(* IEC 61131-3 sources: YaoKangDeviceDemo/src/50_FB, 7 files *)

(* ---- FC_DefaultAxisConfig.st ---- *)
(*============================================================================
  FC_DefaultAxisConfig —— 单轴限位/运动配置工厂默认（P5）
  ----------------------------------------------------------------------------
  返回 Stru_AxisLimitConfig 出厂值。三轴共用同一保守默认，现场按轴调试。
  ⚠ diPulsePerDeg 脉冲当量为占位，必须按 M900 电子齿轮/机械传动比核定后 Save。
==========================================================================*)
FUNCTION FC_DefaultAxisConfig : Stru_AxisLimitConfig

FC_DefaultAxisConfig.rPosLimit     := 90.0;     (* 正限位 ° *)
FC_DefaultAxisConfig.rNegLimit     := -90.0;    (* 负限位 ° *)
FC_DefaultAxisConfig.rInitPos      := 0.0;      (* 初始位置 ° *)
FC_DefaultAxisConfig.rTolerance    := 0.5;      (* 到位容差 ° *)
FC_DefaultAxisConfig.rMaxVel       := 50.0;     (* 最大速度 °/s *)
FC_DefaultAxisConfig.rMinVel       := 0.5;      (* 最小速度 °/s *)
FC_DefaultAxisConfig.rMaxAcc       := 100.0;    (* 最大加速度 °/s² *)
FC_DefaultAxisConfig.rMaxDec       := 100.0;    (* 最大减速度 °/s² *)
FC_DefaultAxisConfig.diPulsePerDeg := 10000;    (* 脉冲当量 Pulse/°（占位，待核定） *)
FC_DefaultAxisConfig.diTimeout     := 30000;    (* 定位超时 ms *)

END_FUNCTION

(* ---- FC_DefaultConditionParams.st ---- *)
(*============================================================================
  FC_DefaultConditionParams —— 调理参数工厂默认（P5）
  ----------------------------------------------------------------------------
  返回一整套 Stru_CondParams 出厂值（三轴 16 段往复 + 全局）。
  ⚠ 默认值仅为安全可校验的保守占位，现场须由工程师按工艺调试后 Save。
  单位：位置 °（脉冲当量见轴 Config）、速度 °/s、加减速 °/s²、时间 ms。
==========================================================================*)
FUNCTION FC_DefaultConditionParams : Stru_CondParams

(*--- 扭腰 SeatTwist：默认单段 ±10°、2 °/s、1 循环 ---*)
FC_DefaultConditionParams.SeatTwist.rAcc             := 20.0;
FC_DefaultConditionParams.SeatTwist.rDec             := 20.0;
FC_DefaultConditionParams.SeatTwist.rInitialPosition := 0.0;
FC_DefaultConditionParams.SeatTwist.iVelocityMode    := 0;
FC_DefaultConditionParams.SeatTwist.iCycleModeLen    := 1;
FC_DefaultConditionParams.SeatTwist.iCycleCount      := -1;
FC_DefaultConditionParams.SeatTwist.iSignalMode      := -1;
FC_DefaultConditionParams.SeatTwist.iSegmentCount    := 1;
FC_DefaultConditionParams.SeatTwist.bEnabled         := TRUE;
FC_DefaultConditionParams.SeatTwist.bOneWay          := FALSE;
FC_DefaultConditionParams.SeatTwist.arPosition[1]    := 10.0;
FC_DefaultConditionParams.SeatTwist.arVelocity[1]    := 2.0;
FC_DefaultConditionParams.SeatTwist.abCycleMode[1]   := FALSE;

(*--- 摆腿 LegAngle：默认单段 +15° ---*)
FC_DefaultConditionParams.LegAngle.rAcc             := 20.0;
FC_DefaultConditionParams.LegAngle.rDec             := 20.0;
FC_DefaultConditionParams.LegAngle.rInitialPosition := 0.0;
FC_DefaultConditionParams.LegAngle.iVelocityMode    := 0;
FC_DefaultConditionParams.LegAngle.iCycleModeLen    := 1;
FC_DefaultConditionParams.LegAngle.iCycleCount      := -1;
FC_DefaultConditionParams.LegAngle.iSignalMode      := -1;
FC_DefaultConditionParams.LegAngle.iSegmentCount    := 1;
FC_DefaultConditionParams.LegAngle.bEnabled         := TRUE;
FC_DefaultConditionParams.LegAngle.bOneWay          := FALSE;
FC_DefaultConditionParams.LegAngle.arPosition[1]    := 15.0;
FC_DefaultConditionParams.LegAngle.arVelocity[1]    := 3.0;
FC_DefaultConditionParams.LegAngle.abCycleMode[1]   := FALSE;

(*--- 冲击 ChestImpact：默认单段 +5°、较快 5 °/s ---*)
FC_DefaultConditionParams.ChestImpact.rAcc             := 30.0;
FC_DefaultConditionParams.ChestImpact.rDec             := 30.0;
FC_DefaultConditionParams.ChestImpact.rInitialPosition := 0.0;
FC_DefaultConditionParams.ChestImpact.iVelocityMode    := 0;
FC_DefaultConditionParams.ChestImpact.iCycleModeLen    := 1;
FC_DefaultConditionParams.ChestImpact.iCycleCount      := -1;
FC_DefaultConditionParams.ChestImpact.iSignalMode      := -1;
FC_DefaultConditionParams.ChestImpact.iSegmentCount    := 1;
FC_DefaultConditionParams.ChestImpact.bEnabled         := TRUE;
FC_DefaultConditionParams.ChestImpact.bOneWay          := FALSE;
FC_DefaultConditionParams.ChestImpact.arPosition[1]    := 5.0;
FC_DefaultConditionParams.ChestImpact.arVelocity[1]    := 5.0;
FC_DefaultConditionParams.ChestImpact.abCycleMode[1]   := FALSE;

(*--- 全局 ---*)
FC_DefaultConditionParams.rPusherPos       := 0.0;      (* 成角目标 °（尾板） *)
FC_DefaultConditionParams.rPusherInitPos   := 0.0;
FC_DefaultConditionParams.diBatchCount     := 1;        (* 老化批次数 *)
FC_DefaultConditionParams.diBatchInterval  := 5000;     (* 批次间隔 ms *)
FC_DefaultConditionParams.diTotalTimeout   := 300000;   (* 总超时 5 min *)
FC_DefaultConditionParams.diConfirmTimeout := 30000;    (* 确认超时 30 s *)
FC_DefaultConditionParams.iCycleCount      := 1;        (* 全局循环次数 *)
FC_DefaultConditionParams.iSignalMode      := 0;        (* 0=脚踏 1=自动 *)

END_FUNCTION

(* ---- FC_DefaultHomingParams.st ---- *)
(*============================================================================
  FC_DefaultHomingParams —— 回零参数工厂默认（P5）
  ----------------------------------------------------------------------------
  返回 Stru_HomingParams 出厂值（普通回零 + 紧急回零 Jog/防夹时序）。
  单位：速度 °/s、加减速 °/s²、扭矩 %、时间 ms。
==========================================================================*)
FUNCTION FC_DefaultHomingParams : Stru_HomingParams

(*--- 限位脱离 ---*)
FC_DefaultHomingParams.rLimitEscapeVel := 2.0;
(*--- 三轴 Jog 速度（内部轴序 1=Chest 2=Seat 3=Leg） ---*)
FC_DefaultHomingParams.rChestJogVel    := 5.0;
FC_DefaultHomingParams.rSeatJogVel     := 5.0;
FC_DefaultHomingParams.rLegJogVel      := 5.0;
(*--- 三轴接近微调（爬行）速度 ---*)
FC_DefaultHomingParams.rChestCrawlVel  := 0.5;
FC_DefaultHomingParams.rSeatCrawlVel   := 0.5;
FC_DefaultHomingParams.rLegCrawlVel    := 0.5;
(*--- 接近区（进入后切爬行） ---*)
FC_DefaultHomingParams.rChestApproachZone := 3.0;
FC_DefaultHomingParams.rSeatApproachZone  := 3.0;
FC_DefaultHomingParams.rLegApproachZone   := 3.0;
(*--- 到位迟滞窗口 ---*)
FC_DefaultHomingParams.rChestHysteresis := 0.3;
FC_DefaultHomingParams.rSeatHysteresis  := 0.3;
FC_DefaultHomingParams.rLegHysteresis   := 0.3;
(*--- Jog 加速度 ---*)
FC_DefaultHomingParams.rChestJogAcc := 20.0;
FC_DefaultHomingParams.rSeatJogAcc  := 20.0;
FC_DefaultHomingParams.rLegJogAcc   := 20.0;
(*--- 防夹扭矩限（净扭矩 %，紧急回零 Jog 超阈即停重试） ---*)
FC_DefaultHomingParams.rAntiPinchTorqueLimit := 40.0;
(*--- 超时/时序 ---*)
FC_DefaultHomingParams.diHomingTimeout         := 60000;   (* 普通回零全流程 60 s *)
FC_DefaultHomingParams.diEmergencyTimeout      := 30000;   (* 紧急回零 30 s *)
FC_DefaultHomingParams.diLimitEscapeTimeout    := 10000;   (* 限位脱离 10 s *)
FC_DefaultHomingParams.diStopReleaseTimeout    := 5000;    (* MC_Stop 释放等待 5 s *)
FC_DefaultHomingParams.diEmergencyCoastMs      := 500;     (* 停后滑行等待 *)
FC_DefaultHomingParams.diEmergencyStallTimeout := 2000;    (* 防夹堵转判定 2 s *)
(*--- 模式/重试 ---*)
FC_DefaultHomingParams.iHomingMode          := 0;         (* 0=顺序 1=并行（默认顺序） *)
FC_DefaultHomingParams.iMaxRetry            := 3;         (* 防夹重试上限 *)
FC_DefaultHomingParams.bEmergencyAllowCalib := FALSE;     (* 紧急回零默认不触发标定 *)

END_FUNCTION

(* ---- FC_DefaultPusherConfig.st ---- *)
(*============================================================================
  FC_DefaultPusherConfig —— 电推杆（尾板）配置工厂默认（P5）
  ----------------------------------------------------------------------------
  返回 Stru_PusherLimitConfig 出厂值：开关型电推杆 + HC_Counter(mm) + 几何解算，
  全部角度阈值直接以 ° 为单位（无脉冲/AD 字段）；堵转/超时/换向缓冲/软限位保留。
  ⚠ 角度°阈值（rMinTravel/rInertiaUp/Down/rStallThreshold）为占位，
    必须现场调试后 Save；几何长度/补偿常量在 GVL_CONST（PUSHER_GEO_*）。
==========================================================================*)
FUNCTION FC_DefaultPusherConfig : Stru_PusherLimitConfig

FC_DefaultPusherConfig.rMaxDeg              := 80.0;     (* 正限位 ° *)
FC_DefaultPusherConfig.rMinDeg              := 0.0;      (* 负限位 ° *)
FC_DefaultPusherConfig.rTolerance           := 0.5;      (* 到位容差 ° *)
FC_DefaultPusherConfig.rInitialPosition     := 0.0;      (* 初始位置（回零目标）° *)
FC_DefaultPusherConfig.rMinTravel           := 2.0;      (* 堵转检测前最小行程 °（占位） *)
FC_DefaultPusherConfig.rHomePosition        := 0.0;      (* 原点位置 ° *)
FC_DefaultPusherConfig.rInertiaUp           := 1.0;      (* 角度增大向惯性补偿 °（占位） *)
FC_DefaultPusherConfig.rInertiaDown         := 1.0;      (* 角度减小向惯性补偿 °（占位） *)
FC_DefaultPusherConfig.rStallThreshold      := 0.5;      (* 堵转位移阈值 °（占位） *)
FC_DefaultPusherConfig.rStallSpeedThreshold := 0.5;      (* 堵转速度阈值 °/s（占位） *)
FC_DefaultPusherConfig.diStallTimeout       := 1000;     (* 堵转判定 1 s *)
FC_DefaultPusherConfig.diTimeout            := 30000;    (* 寻传感器/标定 30 s *)
FC_DefaultPusherConfig.diReverseDelay       := 500;      (* 换向缓冲 0.5 s *)
FC_DefaultPusherConfig.diStopCheck          := 500;      (* 停车滑行等待 0.5 s *)
FC_DefaultPusherConfig.iMaxRetries          := 3;        (* 最大修正次数 *)
FC_DefaultPusherConfig.bInvertPusherDirection := FALSE;  (* 输出方向不取反 *)

END_FUNCTION

(* ---- FC_ValidateParams.st ---- *)
(*============================================================================
  FC_ValidateParams —— 参数 Apply 前校验（P5）
  ----------------------------------------------------------------------------
  对指定参数块的编辑缓冲（HMI 区）做合法性检查，非法即拒绝且不触碰运行区。
  入参：iBlock —— 1=Condition 调理参数（含三轴 16 段往复）
                  2=Pusher 推杆配置（iErrAxis 恒为 AXIS_ID_TAIL=4）
                  3=Chest 冲击轴 Config（iErrAxis=1）
                  4=Leg   转角轴 Config（iErrAxis=2）
                  5=Seat  扭角轴 Config（iErrAxis=3）
                  6=Homing 回零参数（iErrAxis=0，全局）
  出参：iErrCode  —— 0=通过；PARAM_ERR_SEGMENT=1005 段数非法；ERR_PARAM_VALUE=5007 值非法
        iErrAxis  —— 错误所在轴（1=Chest 2=Leg 3=Seat 4=Tail，0=全局）
        iErrField —— 错误字段索引（块内编号，随 iParamErrorField 上报 HMI 定位）
  返回：TRUE=校验通过可 Apply；FALSE=拒绝（三元组已填）。
  说明：仅静态范围/逻辑校验；跨块一致性（如段位置 vs 轴软限位）在运行前检查
       （7xxx，P10）兜底。范围阈值为保守工程值，现场可按工艺收紧。
==========================================================================*)
FUNCTION FC_ValidateParams : BOOL
VAR_INPUT
    iBlock      : INT;
END_VAR
VAR_OUTPUT
    iErrCode    : INT;
    iErrAxis    : INT;
    iErrField   : INT;
END_VAR
(* 段循环下标 vpI 与轴配置视图 vpCfg 为函数私有工作变量，H5U 不支持 FUNCTION 局部
   VAR，已上移为 GVL_Internal 全局（vpI:INT / vpCfg:Stru_AxisLimitConfig）。 *)

(* 默认通过 *)
FC_ValidateParams := TRUE;
iErrCode  := 0;
iErrAxis  := 0;
iErrField := 0;

(*==========================================================================
  iBlock = 1：调理参数（三轴往复 + 全局）
  ==========================================================================*)
IF iBlock = 1 THEN
    (*--- 扭腰 SeatTwist（iErrAxis=AXIS_ID_SEAT=3） ---*)
    IF HMI.Condition.Param.SeatTwist.bEnabled THEN
        IF (HMI.Condition.Param.SeatTwist.iSegmentCount < 1) OR
           (HMI.Condition.Param.SeatTwist.iSegmentCount > 16) THEN
            FC_ValidateParams := FALSE; iErrCode := PARAM_ERR_SEGMENT; iErrAxis := AXIS_ID_SEAT; iErrField := 1; RETURN;
        END_IF;
        IF HMI.Condition.Param.SeatTwist.rAcc <= 0.0 THEN
            FC_ValidateParams := FALSE; iErrCode := ERR_PARAM_VALUE; iErrAxis := AXIS_ID_SEAT; iErrField := 2; RETURN;
        END_IF;
        IF HMI.Condition.Param.SeatTwist.rDec <= 0.0 THEN
            FC_ValidateParams := FALSE; iErrCode := ERR_PARAM_VALUE; iErrAxis := AXIS_ID_SEAT; iErrField := 3; RETURN;
        END_IF;
        IF (HMI.Condition.Param.SeatTwist.iCycleModeLen < 1) OR
           (HMI.Condition.Param.SeatTwist.iCycleModeLen > 16) THEN
            FC_ValidateParams := FALSE; iErrCode := ERR_PARAM_VALUE; iErrAxis := AXIS_ID_SEAT; iErrField := 4; RETURN;
        END_IF;
        FOR vpI := 0 TO HMI.Condition.Param.SeatTwist.iSegmentCount - 1 DO
            IF HMI.Condition.Param.SeatTwist.arVelocity[vpI] <= 0.0 THEN
                FC_ValidateParams := FALSE; iErrCode := ERR_PARAM_VALUE; iErrAxis := AXIS_ID_SEAT; iErrField := 101 + vpI; RETURN;
            END_IF;
        END_FOR;
    END_IF;

    (*--- 摆腿 LegAngle（iErrAxis=AXIS_ID_LEG=2） ---*)
    IF HMI.Condition.Param.LegAngle.bEnabled THEN
        IF (HMI.Condition.Param.LegAngle.iSegmentCount < 1) OR
           (HMI.Condition.Param.LegAngle.iSegmentCount > 16) THEN
            FC_ValidateParams := FALSE; iErrCode := PARAM_ERR_SEGMENT; iErrAxis := AXIS_ID_LEG; iErrField := 1; RETURN;
        END_IF;
        IF HMI.Condition.Param.LegAngle.rAcc <= 0.0 THEN
            FC_ValidateParams := FALSE; iErrCode := ERR_PARAM_VALUE; iErrAxis := AXIS_ID_LEG; iErrField := 2; RETURN;
        END_IF;
        IF HMI.Condition.Param.LegAngle.rDec <= 0.0 THEN
            FC_ValidateParams := FALSE; iErrCode := ERR_PARAM_VALUE; iErrAxis := AXIS_ID_LEG; iErrField := 3; RETURN;
        END_IF;
        IF (HMI.Condition.Param.LegAngle.iCycleModeLen < 1) OR
           (HMI.Condition.Param.LegAngle.iCycleModeLen > 16) THEN
            FC_ValidateParams := FALSE; iErrCode := ERR_PARAM_VALUE; iErrAxis := AXIS_ID_LEG; iErrField := 4; RETURN;
        END_IF;
        FOR vpI := 0 TO HMI.Condition.Param.LegAngle.iSegmentCount - 1 DO
            IF HMI.Condition.Param.LegAngle.arVelocity[vpI] <= 0.0 THEN
                FC_ValidateParams := FALSE; iErrCode := ERR_PARAM_VALUE; iErrAxis := AXIS_ID_LEG; iErrField := 101 + vpI; RETURN;
            END_IF;
        END_FOR;
    END_IF;

    (*--- 冲击 ChestImpact（iErrAxis=AXIS_ID_CHEST=1） ---*)
    IF HMI.Condition.Param.ChestImpact.bEnabled THEN
        IF (HMI.Condition.Param.ChestImpact.iSegmentCount < 1) OR
           (HMI.Condition.Param.ChestImpact.iSegmentCount > 16) THEN
            FC_ValidateParams := FALSE; iErrCode := PARAM_ERR_SEGMENT; iErrAxis := AXIS_ID_CHEST; iErrField := 1; RETURN;
        END_IF;
        IF HMI.Condition.Param.ChestImpact.rAcc <= 0.0 THEN
            FC_ValidateParams := FALSE; iErrCode := ERR_PARAM_VALUE; iErrAxis := AXIS_ID_CHEST; iErrField := 2; RETURN;
        END_IF;
        IF HMI.Condition.Param.ChestImpact.rDec <= 0.0 THEN
            FC_ValidateParams := FALSE; iErrCode := ERR_PARAM_VALUE; iErrAxis := AXIS_ID_CHEST; iErrField := 3; RETURN;
        END_IF;
        IF (HMI.Condition.Param.ChestImpact.iCycleModeLen < 1) OR
           (HMI.Condition.Param.ChestImpact.iCycleModeLen > 16) THEN
            FC_ValidateParams := FALSE; iErrCode := ERR_PARAM_VALUE; iErrAxis := AXIS_ID_CHEST; iErrField := 4; RETURN;
        END_IF;
        FOR vpI := 0 TO HMI.Condition.Param.ChestImpact.iSegmentCount - 1 DO
            IF HMI.Condition.Param.ChestImpact.arVelocity[vpI] <= 0.0 THEN
                FC_ValidateParams := FALSE; iErrCode := ERR_PARAM_VALUE; iErrAxis := AXIS_ID_CHEST; iErrField := 101 + vpI; RETURN;
            END_IF;
        END_FOR;
    END_IF;

    (*--- 全局字段（iErrAxis=0） ---*)
    IF HMI.Condition.Param.diBatchCount < 1 THEN
        FC_ValidateParams := FALSE; iErrCode := ERR_PARAM_VALUE; iErrAxis := 0; iErrField := 10; RETURN;
    END_IF;
    IF HMI.Condition.Param.diBatchInterval < 0 THEN
        FC_ValidateParams := FALSE; iErrCode := ERR_PARAM_VALUE; iErrAxis := 0; iErrField := 11; RETURN;
    END_IF;
    IF HMI.Condition.Param.diTotalTimeout <= 0 THEN
        FC_ValidateParams := FALSE; iErrCode := ERR_PARAM_VALUE; iErrAxis := 0; iErrField := 12; RETURN;
    END_IF;
    IF HMI.Condition.Param.iCycleCount < 1 THEN
        FC_ValidateParams := FALSE; iErrCode := ERR_PARAM_VALUE; iErrAxis := 0; iErrField := 13; RETURN;
    END_IF;
    IF (HMI.Condition.Param.iSignalMode < 0) OR (HMI.Condition.Param.iSignalMode > 1) THEN
        FC_ValidateParams := FALSE; iErrCode := ERR_PARAM_VALUE; iErrAxis := 0; iErrField := 14; RETURN;
    END_IF;

(*==========================================================================
  iBlock = 2：推杆配置（iErrAxis=AXIS_ID_TAIL=4）
  ==========================================================================*)
ELSIF iBlock = 2 THEN
    IF HMI.TailTilt.Config.rMaxDeg <= HMI.TailTilt.Config.rMinDeg THEN
        FC_ValidateParams := FALSE; iErrCode := ERR_PARAM_VALUE; iErrAxis := AXIS_ID_TAIL; iErrField := 1; RETURN;
    END_IF;
    IF HMI.TailTilt.Config.rTolerance <= 0.0 THEN
        FC_ValidateParams := FALSE; iErrCode := ERR_PARAM_VALUE; iErrAxis := AXIS_ID_TAIL; iErrField := 2; RETURN;
    END_IF;
    IF HMI.TailTilt.Config.diTimeout <= 0 THEN
        FC_ValidateParams := FALSE; iErrCode := ERR_PARAM_VALUE; iErrAxis := AXIS_ID_TAIL; iErrField := 3; RETURN;
    END_IF;
    IF HMI.TailTilt.Config.diStallTimeout <= 0 THEN
        FC_ValidateParams := FALSE; iErrCode := ERR_PARAM_VALUE; iErrAxis := AXIS_ID_TAIL; iErrField := 4; RETURN;
    END_IF;
    IF HMI.TailTilt.Config.iMaxRetries < 0 THEN
        FC_ValidateParams := FALSE; iErrCode := ERR_PARAM_VALUE; iErrAxis := AXIS_ID_TAIL; iErrField := 5; RETURN;
    END_IF;
    IF HMI.TailTilt.Config.rStallThreshold <= 0.0 THEN
        FC_ValidateParams := FALSE; iErrCode := ERR_PARAM_VALUE; iErrAxis := AXIS_ID_TAIL; iErrField := 6; RETURN;
    END_IF;
    IF HMI.TailTilt.Config.rMinTravel < 0.0 THEN
        FC_ValidateParams := FALSE; iErrCode := ERR_PARAM_VALUE; iErrAxis := AXIS_ID_TAIL; iErrField := 7; RETURN;
    END_IF;
    IF (HMI.TailTilt.Config.rInitialPosition < HMI.TailTilt.Config.rMinDeg) OR
       (HMI.TailTilt.Config.rInitialPosition > HMI.TailTilt.Config.rMaxDeg) THEN
        FC_ValidateParams := FALSE; iErrCode := ERR_PARAM_VALUE; iErrAxis := AXIS_ID_TAIL; iErrField := 8; RETURN;
    END_IF;
    IF HMI.TailTilt.Config.diReverseDelay < 0 THEN
        FC_ValidateParams := FALSE; iErrCode := ERR_PARAM_VALUE; iErrAxis := AXIS_ID_TAIL; iErrField := 9; RETURN;
    END_IF;

(*==========================================================================
  iBlock = 3/4/5：单轴 Config（Chest=1 / Leg=2 / Seat=3）
  ==========================================================================*)
ELSIF (iBlock = 3) OR (iBlock = 4) OR (iBlock = 5) THEN
    IF iBlock = 3 THEN
        vpCfg := HMI.ChestImpact.Config;  iErrAxis := AXIS_ID_CHEST;
    ELSIF iBlock = 4 THEN
        vpCfg := HMI.LegAngle.Config;     iErrAxis := AXIS_ID_LEG;
    ELSE
        vpCfg := HMI.SeatTwist.Config;    iErrAxis := AXIS_ID_SEAT;
    END_IF;

    IF vpCfg.rPosLimit <= vpCfg.rNegLimit THEN
        FC_ValidateParams := FALSE; iErrCode := ERR_PARAM_VALUE; iErrField := 1; RETURN;
    END_IF;
    IF vpCfg.rTolerance <= 0.0 THEN
        FC_ValidateParams := FALSE; iErrCode := ERR_PARAM_VALUE; iErrField := 2; RETURN;
    END_IF;
    IF vpCfg.rMaxVel <= 0.0 THEN
        FC_ValidateParams := FALSE; iErrCode := ERR_PARAM_VALUE; iErrField := 3; RETURN;
    END_IF;
    IF vpCfg.rMinVel < 0.0 THEN
        FC_ValidateParams := FALSE; iErrCode := ERR_PARAM_VALUE; iErrField := 4; RETURN;
    END_IF;
    IF vpCfg.rMaxVel <= vpCfg.rMinVel THEN
        FC_ValidateParams := FALSE; iErrCode := ERR_PARAM_VALUE; iErrField := 5; RETURN;
    END_IF;
    IF vpCfg.rMaxAcc <= 0.0 THEN
        FC_ValidateParams := FALSE; iErrCode := ERR_PARAM_VALUE; iErrField := 6; RETURN;
    END_IF;
    IF vpCfg.rMaxDec <= 0.0 THEN
        FC_ValidateParams := FALSE; iErrCode := ERR_PARAM_VALUE; iErrField := 7; RETURN;
    END_IF;
    IF vpCfg.diPulsePerDeg <= 0 THEN
        FC_ValidateParams := FALSE; iErrCode := ERR_PARAM_VALUE; iErrField := 8; RETURN;
    END_IF;
    IF vpCfg.diTimeout <= 0 THEN
        FC_ValidateParams := FALSE; iErrCode := ERR_PARAM_VALUE; iErrField := 9; RETURN;
    END_IF;
    IF (vpCfg.rInitPos < vpCfg.rNegLimit) OR (vpCfg.rInitPos > vpCfg.rPosLimit) THEN
        FC_ValidateParams := FALSE; iErrCode := ERR_PARAM_VALUE; iErrField := 10; RETURN;
    END_IF;

(*==========================================================================
  iBlock = 6：回零参数（iErrAxis=0 全局）
  ==========================================================================*)
ELSIF iBlock = 6 THEN
    IF HMI.HomingParams.Params.rLimitEscapeVel <= 0.0 THEN
        FC_ValidateParams := FALSE; iErrCode := ERR_PARAM_VALUE; iErrAxis := 0; iErrField := 1; RETURN;
    END_IF;
    IF HMI.HomingParams.Params.rChestJogVel <= 0.0 THEN
        FC_ValidateParams := FALSE; iErrCode := ERR_PARAM_VALUE; iErrAxis := 0; iErrField := 2; RETURN;
    END_IF;
    IF HMI.HomingParams.Params.rLegJogVel <= 0.0 THEN
        FC_ValidateParams := FALSE; iErrCode := ERR_PARAM_VALUE; iErrAxis := 0; iErrField := 3; RETURN;
    END_IF;
    IF HMI.HomingParams.Params.rSeatJogVel <= 0.0 THEN
        FC_ValidateParams := FALSE; iErrCode := ERR_PARAM_VALUE; iErrAxis := 0; iErrField := 4; RETURN;
    END_IF;
    IF HMI.HomingParams.Params.rChestCrawlVel <= 0.0 THEN
        FC_ValidateParams := FALSE; iErrCode := ERR_PARAM_VALUE; iErrAxis := 0; iErrField := 5; RETURN;
    END_IF;
    IF HMI.HomingParams.Params.rLegCrawlVel <= 0.0 THEN
        FC_ValidateParams := FALSE; iErrCode := ERR_PARAM_VALUE; iErrAxis := 0; iErrField := 6; RETURN;
    END_IF;
    IF HMI.HomingParams.Params.rSeatCrawlVel <= 0.0 THEN
        FC_ValidateParams := FALSE; iErrCode := ERR_PARAM_VALUE; iErrAxis := 0; iErrField := 7; RETURN;
    END_IF;
    IF HMI.HomingParams.Params.rAntiPinchTorqueLimit <= 0.0 THEN
        FC_ValidateParams := FALSE; iErrCode := ERR_PARAM_VALUE; iErrAxis := 0; iErrField := 8; RETURN;
    END_IF;
    IF HMI.HomingParams.Params.diHomingTimeout <= 0 THEN
        FC_ValidateParams := FALSE; iErrCode := ERR_PARAM_VALUE; iErrAxis := 0; iErrField := 9; RETURN;
    END_IF;
    IF HMI.HomingParams.Params.diEmergencyTimeout <= 0 THEN
        FC_ValidateParams := FALSE; iErrCode := ERR_PARAM_VALUE; iErrAxis := 0; iErrField := 10; RETURN;
    END_IF;
    IF HMI.HomingParams.Params.diLimitEscapeTimeout <= 0 THEN
        FC_ValidateParams := FALSE; iErrCode := ERR_PARAM_VALUE; iErrAxis := 0; iErrField := 11; RETURN;
    END_IF;
    IF HMI.HomingParams.Params.diStopReleaseTimeout <= 0 THEN
        FC_ValidateParams := FALSE; iErrCode := ERR_PARAM_VALUE; iErrAxis := 0; iErrField := 12; RETURN;
    END_IF;
    IF HMI.HomingParams.Params.diEmergencyStallTimeout <= 0 THEN
        FC_ValidateParams := FALSE; iErrCode := ERR_PARAM_VALUE; iErrAxis := 0; iErrField := 13; RETURN;
    END_IF;
    IF HMI.HomingParams.Params.iMaxRetry < 0 THEN
        FC_ValidateParams := FALSE; iErrCode := ERR_PARAM_VALUE; iErrAxis := 0; iErrField := 14; RETURN;
    END_IF;
    (*--- 爬行速度必须低于 Jog 速度（四段式减速逻辑前提） ---*)
    IF HMI.HomingParams.Params.rChestCrawlVel >= HMI.HomingParams.Params.rChestJogVel THEN
        FC_ValidateParams := FALSE; iErrCode := ERR_PARAM_VALUE; iErrAxis := 0; iErrField := 15; RETURN;
    END_IF;
    IF HMI.HomingParams.Params.rLegCrawlVel >= HMI.HomingParams.Params.rLegJogVel THEN
        FC_ValidateParams := FALSE; iErrCode := ERR_PARAM_VALUE; iErrAxis := 0; iErrField := 16; RETURN;
    END_IF;
    IF HMI.HomingParams.Params.rSeatCrawlVel >= HMI.HomingParams.Params.rSeatJogVel THEN
        FC_ValidateParams := FALSE; iErrCode := ERR_PARAM_VALUE; iErrAxis := 0; iErrField := 17; RETURN;
    END_IF;
    (*--- 接近区/迟滞必须为正 ---*)
    IF (HMI.HomingParams.Params.rChestApproachZone <= 0.0) OR
       (HMI.HomingParams.Params.rLegApproachZone   <= 0.0) OR
       (HMI.HomingParams.Params.rSeatApproachZone  <= 0.0) THEN
        FC_ValidateParams := FALSE; iErrCode := ERR_PARAM_VALUE; iErrAxis := 0; iErrField := 18; RETURN;
    END_IF;
    IF (HMI.HomingParams.Params.rChestHysteresis <= 0.0) OR
       (HMI.HomingParams.Params.rLegHysteresis   <= 0.0) OR
       (HMI.HomingParams.Params.rSeatHysteresis  <= 0.0) THEN
        FC_ValidateParams := FALSE; iErrCode := ERR_PARAM_VALUE; iErrAxis := 0; iErrField := 19; RETURN;
    END_IF;

ELSE
    (* 未知块号：直接拒绝 *)
    FC_ValidateParams := FALSE; iErrCode := ERR_PARAM_VALUE; iErrAxis := 0; iErrField := 0;
END_IF;

END_FUNCTION

(* ---- FB_AxisControl.st ---- *)
(*============================================================================
  FB_AxisControl —— 单轴伺服控制（M900，EtherCAT / CiA402），三轴各实例化一个
  ----------------------------------------------------------------------------
  平台事实（汇川 H5U / InoProShop，旧工程变量表导出佐证）：
    EtherCAT 轴引用 AXIS_REF（底层 _sMCAXIS_INFO）为结构体，直接写字段即下发命令：
      bPowerOn 使能 | bReset 复位 | bStop 停止 | bHome 原点回归 | bSetPos 设当前位
      bJogP/bJogN 点动± | bAbsPos 绝对定位 | bRelPos 相对定位 | bRevPos 往复
      fJogVelocity 点动速度 | fTarPosition1/fTarVelocity1/fTarAcceleration1/
      fTarDecelaration1/wCurveType1 目标位置/速度/加减速/曲线
    直接读字段取状态：
      bPowerState 已使能 | bMotionState 运动中 | bphlimit/bnhlimit 硬件±限位
      bpslimit/bnslimit 软件±限位 | bhomestate 原点开关 | wPLCOpenState PLCopen 状态
      fActPosition/fActVelocity/fActTorque 实际位置/速度/力矩
      wServoError 驱动器故障 | wAxisError 轴故障 | fFollowPos 跟随误差
  职责（P7）：
    - 运动状态机：IDLE/ENABLING/READY/JOG/MOVE/BUFFER/ERROR；
    - 点动（电平，限位方向禁动）、绝对/相对定位（脉冲触发，软限位校验）、
      16 段缓冲（MoveBuffer，逐段绝对定位，P10 调理联动用）；
    - 到位/在初始位/静止判定；步骤超时（2005）；驱动器故障（2001，子码=Er.xxx）；
      未使能/未参考定位拒绝（2006）；软限位拒绝（2004）；
    - 力估算：静止扭矩基线学习、净扭矩、牵引力 N（低通）、超力实时态/锁存
      （锁存供 SAFETY 保护停机，事件 1206 由 SAFETY_MANAGER 统一提交，本 FB 不报）。
  单写源：本 FB 仅在 PRG_OutputAdapter（扫描链第 10 环）内实例化调用，
          是轴命令字段与轴 Status 镜像的唯一写入点。
  时间基准：扫描周期按 10ms 计（任务组态确认后统一修正），超时/持续用 diScanCount 推算。
  ----------------------------------------------------------------------------
  变量表导入说明（汇川 InoProShop）：
  接口表 FB_AxisControl_new.csv 已含全部 66 个引脚（含 Axis / stStatus），文件编码必须为
  UTF-16 LE + BOM（汇川原生导出格式；UTF-8 会导入失败），可直接导入、无需手动新建引脚。
  结构体/轴引用引脚均按单行写法（不展开子字段），已验证可正常导入。导入后仅需：
    ① Axis : AXIS_REF（VAR_INPUT）—— 引脚随 CSV 自动创建；在【实例化调用处】把本输入
       绑定到轴组态对应轴：Axis_胸背 / Axis_臀盘 / Axis_臀腿。
    ② stStatus : Stru_AxisStatus（VAR_OUTPUT）—— 自定义结构体（UDT），导入前须先把类型
       定义加入工程（src\00_Globals\ST_StruHMI.st：Stru_AxisStatus L479，成员
       Servo:Stru_ServoAxisStatus L429 / Force:Stru_AxisForceStatus L461）。
==========================================================================*)
FUNCTION_BLOCK FB_AxisControl
VAR_INPUT
    (* 轴引用引脚：随 FB_AxisControl_new.csv（UTF-16 LE）导入自动创建，无需手动新建；
       实例化调用时把本输入绑定到轴组态对应轴：Axis_胸背/臀盘/臀腿（底层 _sMCAXIS_INFO） *)
    Axis            : AXIS_REF;         (* EtherCAT 轴引用（Axis_胸背/臀盘/臀腿） *)
    iAxisId         : INT;              (* 轴编号（AXIS_ID_CHEST/SEAT/LEG，故障定位） *)
    bEnable         : BOOL;             (* 使能电平（源：POWER 分时上电 axisPowerEnable） *)
    bReset          : BOOL;             (* 复位轴错误（脉冲） *)
    bZeroComm       : BOOL;             (* 原点标定（脉冲，仅工厂建零，MC_Home） *)
    bStop           : BOOL;             (* 立即减速停车（电平，含安全链） *)
    bMoveAbs        : BOOL;             (* 绝对定位（脉冲） *)
    bMoveRel        : BOOL;             (* 相对定位（脉冲） *)
    bJogPos         : BOOL;             (* 正向点动（电平） *)
    bJogNeg         : BOOL;             (* 负向点动（电平） *)
    bMoveBuffer     : BOOL;             (* 16 段缓冲启动（脉冲，P10 联动） *)
    arSegPos        : REAL[16];         (* 缓冲段目标位置表 *)
    arSegVel        : REAL[16];         (* 缓冲段目标速度表 *)
    iSegCount       : INT;              (* 缓冲段数（1..16） *)
    rTargetPos      : REAL;             (* 单段目标位置 *)
    rTargetVel      : REAL;             (* 单段目标速度 *)
    rJogVel         : REAL;             (* 点动速度 *)
    rAcc            : REAL;             (* 加速度 *)
    rDec            : REAL;             (* 减速度 *)
    rInitPos        : REAL;             (* 初始位置（bAtInit 判定基准） *)
    rPosLimit       : REAL;             (* 正软限位 *)
    rNegLimit       : REAL;             (* 负软限位 *)
    rTolerance      : REAL;             (* 到位/在初始位容差 *)
    diTimeout       : DINT;             (* 单段定位超时 (ms) *)
    bSafetyStop     : BOOL;             (* 安全链停车（硬/软急停/保护停机/硬限位） *)
    bZeroCommRetain : BOOL;             (* 建零标志镜像（retainZeroComm[i]，P9 写） *)
    bLearnBias      : BOOL;             (* 学习静止扭矩基线（脉冲） *)
    rForceScaleN    : REAL;             (* 净扭矩%→牵引力 N 换算系数（台架标定） *)
    rOverForceN     : REAL;             (* 超力阈值 (N，低通后) *)
END_VAR
VAR_OUTPUT
    (* 结构体引脚：随 FB_AxisControl_new.csv（UTF-16 LE）导入自动创建，无需手动新建；
       导入前须先把类型 Stru_AxisStatus 加入工程（ST_StruHMI.st L479，
       成员 Servo:Stru_ServoAxisStatus L429 / Force:Stru_AxisForceStatus L461） *)
    stStatus        : Stru_AxisStatus;  (* 轴状态全量镜像（→ HMI.<Axis>.Status） *)
    bFaultEvent     : BOOL;             (* 本扫新故障事件脉冲（→ OUTPUT_ADAPTER 序列化提交） *)
    iFaultCode      : INT;              (* 故障码（2xxx） *)
    iFaultLevel     : INT;              (* 级别 1=Warning 2=Critical *)
    iFaultSub       : INT;              (* 子码（驱动器 Er.xxx） *)
END_VAR
VAR
    iStep           : INT;              (* 运动状态机 AXST_* *)
    iBufSeg         : INT;              (* 缓冲当前段（1..iSegCount） *)
    bMoving         : BOOL;             (* 定位/缓冲进行中 *)
    bJogActive      : BOOL;             (* 点动进行中 *)
    rLastTarget     : REAL;             (* 本段目标位置（到位判定） *)
    diMoveSnap      : DINT;             (* 本段启动扫描计数（超时判定，跨段每段重置） *)
    diMoveStartSnap : DINT;             (* 本次离散定位整体启动扫描计数（用时锁存，跨段不重置） *)
    diMoveTimeLatch : DINT;             (* 最近一次离散定位完成用时 (ms)，完成时锁存 *)
    diOverCnt       : DINT;             (* 超力持续扫描计数（×10ms） *)
    rBiasP          : REAL;             (* 正侧静止基线 (%) *)
    rBiasN          : REAL;             (* 负侧静止基线 (%) *)
    bBiasPValid     : BOOL;
    bBiasNValid     : BOOL;
    rFiltN          : REAL;             (* 牵引力低通值 (N) *)
    bDrvErrPrev     : BOOL;             (* 驱动器故障锁存（事件边沿用） *)
    bEncFltMatch    : BOOL;             (* 本扫驱动器码命中编码器反馈类报警（联调填码） *)
    bEncFltLatch    : BOOL;             (* 编码器故障锁存（bReset 清除，绝对位置不可信） *)
    bOverLatch      : BOOL;             (* 超力锁存（bReset 清除） *)
    bToutReported   : BOOL;             (* 本段超时已报（防重复） *)
    rActPos         : REAL;
    rActVel         : REAL;
    rActTorque      : REAL;
    bPowerState     : BOOL;
    bMotionState    : BOOL;
    bDrvErr         : BOOL;
    iDrvCode        : INT;
    bStandStill     : BOOL;
    bAtInit         : BOOL;
    bInPosition     : BOOL;
    rNetPct         : REAL;
    rForceRawN      : REAL;
    bOverForce      : BOOL;
    bSwRej          : BOOL;             (* 本扫软限位/非法拒绝事件 *)
    iRejCode        : INT;
    bTimeoutEv      : BOOL;             (* 本扫超时事件 *)
    iTimeoutCode    : INT;
END_VAR

(*------------------------------------------------------------
  1) 驱动器状态采集（每扫直读轴字段）
------------------------------------------------------------*)
rActPos      := Axis.fActPosition;
rActVel      := Axis.fActVelocity;
rActTorque   := Axis.fActTorque;
bPowerState  := Axis.bPowerState;
bMotionState := Axis.bMotionState;
iDrvCode     := Axis.wServoError;
IF (Axis.wServoError <> 0) OR (Axis.wAxisError <> 0) THEN
    bDrvErr := TRUE;
    IF Axis.wServoError <> 0 THEN
        iDrvCode := Axis.wServoError;
    ELSE
        iDrvCode := Axis.wAxisError;
    END_IF;
ELSE
    bDrvErr := FALSE;
END_IF;

(* 1.1 编码器反馈故障：iDrvCode 命中 M900 编码器/反馈类报警码即视为绝对位置不可信。
       → 置 stStatus.Servo.bEncoderFault，下游 SAFETY 保护停机并报 ERR_AXIS_ENCODER(2002)。
       TODO 联调：M900(CiA402/EtherCAT) 编码器反馈类报警 Er.xxx 确切码表需依驱动器手册
                  及台架实测填入下面判定（文档仅有的 Er.101/201/234 为 SV630 举例，不可套用）。
                  填码前默认不命中（bEncFltMatch:=FALSE），编码器故障链保持断开、不误保护。 *)
bEncFltMatch := FALSE;
(* 联调填码示例（待手册/台架确认后启用，并保留有效码）：
   bEncFltMatch := bDrvErr AND ( (iDrvCode = ErXXX) OR (iDrvCode = ErYYY) ... );
   （编码器断线/多圈电池掉电/反馈计数异常等均属此列；命中后绝对位置不可信，禁定位） *)

(* 锁存：命中即置位保持；复位脉冲且驱动器故障已消时清除（与 bToutReported 同步复位） *)
IF bEncFltMatch THEN
    bEncFltLatch := TRUE;
END_IF;

(* 静止：已使能且非运动态（速度窗由驱动器 bMotionState 保证） *)
bStandStill := bPowerState AND NOT bMotionState;
bAtInit     := bPowerState AND (ABS(rActPos - rInitPos) <= rTolerance);

(*------------------------------------------------------------
  2) 默认输出与事件清零（每扫先清零，按条件再置位）
------------------------------------------------------------*)
bFaultEvent  := FALSE;
iFaultCode   := 0;
iFaultLevel  := 0;
iFaultSub    := 0;
bSwRej       := FALSE;
iRejCode     := 0;
bTimeoutEv   := FALSE;
iTimeoutCode := 0;

Axis.bPowerOn := bEnable;          (* 使能电平直写（POWER 已按急停/时序裁决） *)
Axis.bJogP    := FALSE;
Axis.bJogN    := FALSE;
Axis.bAbsPos  := FALSE;
Axis.bRelPos  := FALSE;
Axis.bStop    := FALSE;
Axis.bReset   := bReset;           (* 复位脉冲直透（驱动器清错） *)
Axis.bHome    := FALSE;

(*------------------------------------------------------------
  3) 故障/复位处理
------------------------------------------------------------*)
(* 3.1 驱动器故障上升沿 → 2001 Critical，子码=驱动器 Er.xxx *)
IF bDrvErr AND NOT bDrvErrPrev THEN
    bFaultEvent := TRUE;
    iFaultCode  := ERR_AXIS_DRIVE;
    iFaultLevel := 2;
    iFaultSub   := iDrvCode;
END_IF;
bDrvErrPrev := bDrvErr;

(* 3.2 复位脉冲且驱动器故障已消 → 清锁存 *)
IF bReset AND NOT bDrvErr THEN
    bOverLatch    := FALSE;
    bToutReported := FALSE;
    bEncFltLatch  := FALSE;
    IF iStep = AXST_ERROR THEN
        iStep := AXST_READY;
    END_IF;
END_IF;

IF bDrvErr THEN
    iStep := AXST_ERROR;
END_IF;

(*------------------------------------------------------------
  4) 力估算（每扫）
------------------------------------------------------------*)
(* 4.1 基线学习：静止时收到学习脉冲，记录当前力矩为正/负侧基线 *)
IF bLearnBias AND bStandStill THEN
    rBiasP      := rActTorque;
    rBiasN      := rActTorque;
    bBiasPValid := TRUE;
    bBiasNValid := TRUE;
END_IF;

(* 4.2 净扭矩：按运动方向选侧基线；静止未学基线时净力按 0 *)
IF bMotionState THEN
    IF rActVel >= 0 THEN
        IF bBiasPValid THEN
            rNetPct := rActTorque - rBiasP;
        ELSE
            rNetPct := 0.0;
        END_IF;
    ELSE
        IF bBiasNValid THEN
            rNetPct := rActTorque - rBiasN;
        ELSE
            rNetPct := 0.0;
        END_IF;
    END_IF;
ELSE
    rNetPct := 0.0;
END_IF;
rForceRawN := ABS(rNetPct) * rForceScaleN;

(* 4.3 一阶低通（系数 FORCE_LPF_ALPHA，台架可标） *)
rFiltN := rFiltN + (rForceRawN - rFiltN) * FORCE_LPF_ALPHA;

(* 4.4 超力：运动中低通值超阈持续 OVERFORCE_SCAN 扫（≈500ms@10ms）→ 锁存 *)
bOverForce := bMotionState AND bBiasPValid AND (rFiltN > rOverForceN);
IF bOverForce THEN
    diOverCnt := diOverCnt + 1;
    IF diOverCnt >= OVERFORCE_SCAN THEN
        bOverLatch := TRUE;
    END_IF;
ELSE
    diOverCnt := 0;
END_IF;

(*------------------------------------------------------------
  5) 运动状态机（无驱动器故障时才接受运动命令）
------------------------------------------------------------*)
IF NOT bDrvErr THEN
    (* 5.1 使能态迁移 *)
    IF NOT bPowerState THEN
        IF bEnable THEN
            iStep := AXST_ENABLING;
        ELSE
            iStep := AXST_IDLE;
            bMoving    := FALSE;
            bJogActive := FALSE;
        END_IF;
    ELSIF iStep <> AXST_MOVE AND iStep <> AXST_BUFFER AND iStep <> AXST_JOG THEN
        iStep := AXST_READY;
    END_IF;

    (* 5.2 原点标定（工厂建零）：已使能才发 MC_Home，其余门控在 P9 任务层 *)
    IF bZeroComm AND bPowerState THEN
        Axis.bHome := TRUE;
    END_IF;

    (* 5.3 停车（安全链/停止命令）：撤掉所有运动命令，发 bStop 脉冲 *)
    IF bStop OR bSafetyStop THEN
        Axis.bStop    := TRUE;
        Axis.bJogP    := FALSE;
        Axis.bJogN    := FALSE;
        bMoving       := FALSE;
        bJogActive    := FALSE;
        iStep         := AXST_READY;
        bToutReported := TRUE;   (* 中断的段不再报超时 *)
    ELSIF bPowerState THEN
        (* 5.4 点动（电平）：限位方向禁动（防冲出软限位） *)
        IF bJogPos AND (rActPos < rPosLimit) AND NOT bMoving THEN
            Axis.bJogP       := TRUE;
            Axis.fJogVelocity:= rJogVel;
            bJogActive       := TRUE;
            iStep            := AXST_JOG;
        ELSIF bJogNeg AND (rActPos > rNegLimit) AND NOT bMoving THEN
            Axis.bJogN       := TRUE;
            Axis.fJogVelocity:= rJogVel;
            bJogActive       := TRUE;
            iStep            := AXST_JOG;
        END_IF;
        IF bJogActive AND NOT bJogPos AND NOT bJogNeg THEN
            bJogActive := FALSE;
            IF NOT bMoving THEN
                iStep := AXST_READY;
            END_IF;
        END_IF;

        (* 5.5 绝对/相对/缓冲启动（静止态才接受新段任务） *)
        IF NOT bMoving AND NOT bJogActive THEN
            IF bMoveBuffer AND (iSegCount >= 1) THEN
                (* 缓冲需参考有效（已建零），否则 2006 拒绝 *)
                IF NOT bZeroCommRetain THEN
                    bSwRej := TRUE; iRejCode := ERR_AXIS_CMD_ILLEGAL;
                ELSE
                    (* 首段立即下发绝对定位命令 *)
                    iBufSeg                := 1;
                    Axis.fTarPosition1     := arSegPos[1];
                    Axis.fTarVelocity1     := arSegVel[1];
                    Axis.fTarAcceleration1 := rAcc;
                    Axis.fTarDecelaration1 := rDec;
                    Axis.wCurveType1       := 0;
                    Axis.bAbsPos           := TRUE;
                    rLastTarget            := arSegPos[1];
                    diMoveSnap             := diScanCount;
                    diMoveStartSnap        := diScanCount;
                    diMoveTimeLatch        := 0;
                    bMoving                := TRUE;
                    bToutReported          := FALSE;
                    iStep                  := AXST_BUFFER;
                END_IF;
            ELSIF bMoveAbs THEN
                IF NOT bZeroCommRetain THEN
                    bSwRej := TRUE; iRejCode := ERR_AXIS_CMD_ILLEGAL;     (* 未建零禁绝对定位 *)
                ELSIF (rTargetPos > rPosLimit) OR (rTargetPos < rNegLimit) THEN
                    bSwRej := TRUE; iRejCode := ERR_AXIS_SWLIMIT;        (* 越软限位拒绝 *)
                ELSE
                    Axis.fTarPosition1    := rTargetPos;
                    Axis.fTarVelocity1    := rTargetVel;
                    Axis.fTarAcceleration1:= rAcc;
                    Axis.fTarDecelaration1:= rDec;
                    Axis.wCurveType1      := 0;
                    Axis.bAbsPos          := TRUE;
                    rLastTarget           := rTargetPos;
                    diMoveSnap            := diScanCount;
                    diMoveStartSnap       := diScanCount;
                    diMoveTimeLatch       := 0;
                    bMoving               := TRUE;
                    bToutReported        := FALSE;
                    iStep                 := AXST_MOVE;
                END_IF;
            ELSIF bMoveRel THEN
                (* 相对定位：增量运动，仍受软限位约束（目标落点校验） *)
                IF (rActPos + rTargetPos > rPosLimit) OR (rActPos + rTargetPos < rNegLimit) THEN
                    bSwRej := TRUE; iRejCode := ERR_AXIS_SWLIMIT;
                ELSE
                    Axis.fTarPosition1    := rTargetPos;
                    Axis.fTarVelocity1    := rTargetVel;
                    Axis.fTarAcceleration1:= rAcc;
                    Axis.fTarDecelaration1:= rDec;
                    Axis.wCurveType1      := 0;
                    Axis.bRelPos          := TRUE;
                    rLastTarget           := rActPos + rTargetPos;
                    diMoveSnap            := diScanCount;
                    diMoveStartSnap       := diScanCount;
                    diMoveTimeLatch       := 0;
                    bMoving               := TRUE;
                    bToutReported        := FALSE;
                    iStep                 := AXST_MOVE;
                END_IF;
            END_IF;
        END_IF;

        (* 5.6 段推进与完成判定（运动中驱动器 bMotionState 回落且到位 → 本段完成） *)
        IF bMoving AND NOT bMotionState AND (ABS(rActPos - rLastTarget) <= rTolerance) THEN
            IF iStep = AXST_BUFFER THEN
                IF iBufSeg < iSegCount THEN
                    (* 下一段：目标/速度取自段表，发绝对定位脉冲 *)
                    iBufSeg               := iBufSeg + 1;
                    Axis.fTarPosition1    := arSegPos[iBufSeg];
                    Axis.fTarVelocity1    := arSegVel[iBufSeg];
                    Axis.fTarAcceleration1:= rAcc;
                    Axis.fTarDecelaration1:= rDec;
                    Axis.wCurveType1      := 0;
                    Axis.bAbsPos          := TRUE;
                    rLastTarget           := arSegPos[iBufSeg];
                    diMoveSnap            := diScanCount;
                    bToutReported        := FALSE;
                ELSE
                    (* 全部段完成：锁存整体离散运动用时（整体起点→末段到位，ms） *)
                    diMoveTimeLatch := (diScanCount - diMoveStartSnap) * 10;
                    bMoving := FALSE;
                    iStep   := AXST_READY;
                END_IF;
            ELSE
                (* 单段完成：锁存本段离散运动用时（ms） *)
                diMoveTimeLatch := (diScanCount - diMoveSnap) * 10;
                bMoving := FALSE;
                iStep   := AXST_READY;
            END_IF;
        END_IF;

        (* 5.7 单段超时：diTimeout(ms) 内未到位 → 2005 Critical，发停车 *)
        IF bMoving AND NOT bToutReported THEN
            IF (diScanCount - diMoveSnap) * 10 >= diTimeout THEN
                bToutReported := TRUE;
                bTimeoutEv    := TRUE;
                iTimeoutCode  := ERR_AXIS_STEP_TOUT;
                Axis.bStop    := TRUE;
                bMoving       := FALSE;
                iStep         := AXST_ERROR;
            END_IF;
        END_IF;
    END_IF;
END_IF;

(* 5.8 拒绝/超时事件上报（驱动器故障事件优先） *)
IF NOT bFaultEvent THEN
    IF bTimeoutEv THEN
        bFaultEvent := TRUE; iFaultCode := iTimeoutCode; iFaultLevel := 2; iFaultSub := 0;
    ELSIF bSwRej THEN
        bFaultEvent := TRUE; iFaultCode := iRejCode; iFaultLevel := 1; iFaultSub := 0;
    END_IF;
END_IF;

(* 到位：静止且在最后目标容差内 *)
bInPosition := bPowerState AND NOT bMotionState AND NOT bMoving
               AND (ABS(rActPos - rLastTarget) <= rTolerance);

(*------------------------------------------------------------
  6) 状态全量回填 stStatus（Servo + Force + 业务层）
------------------------------------------------------------*)
stStatus.Servo.rActPosition         := rActPos;
stStatus.Servo.rActVelocity         := rActVel;
stStatus.Servo.rActTorque           := rActTorque;
stStatus.Servo.iDriveErrorCode      := iDrvCode;
stStatus.Servo.iErrorCode           := iFaultCode;
stStatus.Servo.diDiscreteMotionTime := diMoveTimeLatch;   (* 最近一次离散定位完成用时(ms)，完成时锁存 *)
stStatus.Servo.bEnabled             := bPowerState;
stStatus.Servo.bReady               := bPowerState AND NOT bDrvErr;
stStatus.Servo.bBusy                := bMotionState OR bMoving OR bJogActive;
stStatus.Servo.bDone                := bInPosition;
stStatus.Servo.bStandStill          := bStandStill;
stStatus.Servo.bInPosition          := bInPosition;
stStatus.Servo.bDiscreteMotion      := bMoving;
stStatus.Servo.bMoveDone            := bInPosition AND (iStep = AXST_READY);  (* 完成脉冲近似 *)
stStatus.Servo.bZeroCommissioned    := bZeroCommRetain;
stStatus.Servo.bZeroCommissioning   := bZeroComm;
stStatus.Servo.bOriginSwitch        := Axis.bhomestate;
stStatus.Servo.bPosLimit            := Axis.bphlimit OR Axis.bpslimit;
stStatus.Servo.bNegLimit            := Axis.bnhlimit OR Axis.bnslimit;
stStatus.Servo.bError               := bDrvErr OR (iStep = AXST_ERROR);
stStatus.Servo.bStopping            := bStop OR bSafetyStop OR (Axis.wPLCOpenState = 3);
stStatus.Servo.bEncoderFault        := bEncFltLatch;   (* 编码器反馈故障锁存（码表见 1.1 TODO，联调填码） *)

stStatus.Force.rBiasPosPct          := rBiasP;
stStatus.Force.rBiasNegPct          := rBiasN;
stStatus.Force.rNetTorquePct        := rNetPct;
stStatus.Force.rForceRawN           := rForceRawN;
stStatus.Force.rForceFiltN          := rFiltN;
stStatus.Force.diOverForceET        := diOverCnt * 10;
stStatus.Force.bForceValid          := bPowerState AND (bBiasPValid OR bBiasNValid);
stStatus.Force.bBiasPosValid        := bBiasPValid;
stStatus.Force.bBiasNegValid        := bBiasNValid;
stStatus.Force.bOverForce           := bOverForce;
stStatus.Force.bOverForceLatched    := bOverLatch;

stStatus.iCurrentStep               := iStep;
stStatus.diMotionTime               := (diScanCount - diMoveSnap) * 10;
stStatus.iErrorCode                 := iFaultCode;
stStatus.bCalibrated                := bZeroCommRetain;
stStatus.bError                     := bDrvErr OR (iStep = AXST_ERROR);
stStatus.bWarning                   := bSwRej;
stStatus.bAxisErrorStopping         := bTimeoutEv;
stStatus.bAtInit                    := bAtInit;

END_FUNCTION_BLOCK

(* ---- FB_PusherControl.st ---- *)
(*============================================================================
  FB_PusherControl —— 尾板电推杆控制（开关型，双参考模式）
  ----------------------------------------------------------------------------
  职责：点动/回零/原点标定/自动定位/手动 Preset/回初始位；堵转与超时保护、
        换向缓冲、惯性补偿；双参考 iReferenceMode：
          0 = 脉冲计数 + 原点传感器；1 = AD 三次拟合角度（rFitK0..K3）。
        bHomed 与 bCalibrated 解耦；未校准/参考无效禁自动定位（报 3024）。
  线结构体：HMI.TailTilt.Status/Cmd/Motion/Config/ConfigCmd（字段见 ST_StruHMI.st）。
  物理输出 Q_Pusher_Up/Q_Pusher_Down 经 OUTPUT_ADAPTER 单写；本 FB 出请求位。
  P1：接口骨架。P8：校准流程（3101–3107）、堵转 5001/超时 5002/重试 5003。
==========================================================================*)
FUNCTION_BLOCK FB_PusherControl
VAR_INPUT
    bEnable       : BOOL;            (* 使能 *)
    bJogUp        : BOOL;            (* 上行点动（电平） *)
    bJogDown      : BOOL;            (* 下行点动（电平） *)
    bHome         : BOOL;            (* 回零：移动到原点位置（脉冲） *)
    bCalibrate    : BOOL;            (* 原点标定（脉冲） *)
    bAutoMove     : BOOL;            (* 自动定位到 rTargetAngle（脉冲） *)
    bManualPreset : BOOL;            (* 手动清零/预设（脉冲） *)
    bResetError   : BOOL;            (* 重置故障（脉冲） *)
    bStop         : BOOL;            (* 停止 *)
    rTargetAngle  : REAL;            (* 目标角度 (°) *)
    iReferenceMode: INT;             (* 0=脉冲+原点  1=AD 拟合 *)
    bHomeSwitch   : BOOL;            (* 原点传感器（去抖后 ioPusherOrigin） *)
    diAdRaw       : DINT;            (* AD 原始值 *)
    bAdValid      : BOOL;            (* AD 有效 *)
    bSafetyStop   : BOOL;            (* 安全链停车 *)
END_VAR
VAR_OUTPUT
    bRunUp        : BOOL;            (* 请求上行（→ OUTPUT_ADAPTER → Q_Pusher_Up） *)
    bRunDown      : BOOL;            (* 请求下行 *)
    bBusy         : BOOL;
    bDone         : BOOL;
    bHomed        : BOOL;            (* 已回零（与标定解耦） *)
    bCalibrated   : BOOL;            (* 已校准 *)
    bReferenceValid: BOOL;           (* 坐标参考有效 *)
    bError        : BOOL;
    iErrorCode    : INT;             (* 5001 堵转 / 5002 超时 / 5003 重试超限 / 3024 未校准 *)
    rCurrAngle    : REAL;            (* 当前角度（°） *)
END_VAR
VAR
    iStep         : INT;
    iRetryCount   : INT;
    (* H5U 定时器为内联指令 TONR(IN:=,PT:=,Q=>布尔位)，无需 TON 实例：
       tStepTimer/tStallTimer 即 TONR 的 Q=> 输出 BOOL（定时到标志）。 *)
    tStepTimer    : BOOL;   (* 步序定时到（P8：TONR Q=>tStepTimer） *)
    tStallTimer   : BOOL;   (* 堵转定时到（P8：TONR Q=>tStallTimer） *)
END_VAR

(* TODO P8:
   - 角度源：模式 0 脉冲计数 × rPulsePerDeg；模式 1 AD 三次拟合 K0..K3 + 跳变保护。
   - 校准流程：默认上行找原点；已压原点→先下行脱离→缓冲 diReverseDelay→上行精找→
     30ms 去抖→清零；上行撞顶堵转→缓冲换向→下行反找；全局超时 diTimeout。
   - 堵转：走过 rMinTravel 后，速度趋零持续 diStallTimeout → 5001，换向缓冲后重试，
     超 iMaxRetries → 5003。
   - 自动定位前校验 bCalibrated/bReferenceValid，否则报 3024 拒绝。
   - 惯性补偿 rInertiaUp/Down、软限位 rMaxDeg/rMinDeg、到位容差 rTolerance。
   - 方向取反 bInvertPusherDirection 作用于输出请求位。
   - 状态位全量回写 HMI.TailTilt.Status（bHomeSensorHealthy/StuckOn/StuckOff/
     bHomePlausible/bSensorChecked/bAutoMovePending 等，P9 传感器诊断）。 *)
END_FUNCTION_BLOCK
